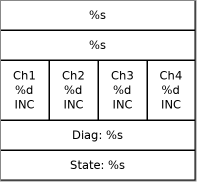
VISUALIZATION TplTsConnectionEL3214  // 197x182
VAR_IN_OUT
	stConnectionDiag 			:FB_TwinSafeConnectionEL3214;
END_VAR
(* End *)
    Rectangle (0,0 195x30), "%s", text variable: stConnectionDiag.sEcSlaveName, colour toggle: stConnectionDiag.sDiag = 'No error'
    Rectangle (0,60 49x60), "Ch1 %d INC", text variable: stConnectionDiag.nInSafeDataValue1
    Rectangle (49,60 49x60), "Ch2 %d INC", text variable: stConnectionDiag.nInSafeDataValue2
    Rectangle (98,60 49x60), "Ch3 %d INC", text variable: stConnectionDiag.nInSafeDataValue3
    Rectangle (147,60 48x60), "Ch4 %d INC", text variable: stConnectionDiag.nInSafeDataValue4
    Rectangle (0,120 195x30), "Diag: %s", text variable: stConnectionDiag.sDiag, colour toggle: stConnectionDiag.sDiag <> 'No error'
    Rectangle (0,150 195x30), "State: %s", text variable: stConnectionDiag.sState
    Rectangle (0,30 195x30), "%s", text variable: stConnectionDiag.sEcSlaveType
END_VISUALIZATION

(* stored: Version 1.1.0.1
   Visu TplTsConnectionEL3214: Id {2f376470-b3af-43cf-be81-bd2a47da1714} *)
